# EPICS autosave request: iocBoot/ioc13idd_LVP/auto_settings.req
file "E1608_settings.req",       P=$(P)MC1:
file "E1608_settings.req",       P=$(P)MC2:
file "Keithley2kDMM_mf10_settings.req", P=$(P), Dmm=DMM3
file "Keithley2kDMM_mf10_settings.req", P=$(P), Dmm=DMM4
file "ID_LVP_pressure_settings.req", P=$(P), R=Press_
file "Galil_settings.req", P=$(MP)
